Omron Sysmac Studio project PC與TCP Socket測試_5 (Sysmac Studio 1.1.7.20, StandardProject)

# Controller new_Controller_0: NJ501-1300 version 1.10
Units and slaves: 電源 : NJ-Px3001; CPU : NJ501-1300
Axis X, settings changed from default: UnitsConversion=EnumElement2, UnitsNumerator=1048576, UnitsDenominator=5, MaxVelocity=250, MaxJogVelocity=250, HomingMode=BackupAndProximitySignalOff, StartDirection=NegativeDirection, OriginInputDetectionDirection=NegativeDirection, HomingVelocity=50, HomingApproachVelocity=25, CompensationVelocity=25
Axis Y, settings changed from default: AxisNumber=1, UnitsConversion=EnumElement2, UnitsNumerator=1048576, UnitsDenominator=5, MaxVelocity=250, MaxJogVelocity=250, HomingMode=BackupAndProximitySignalOff, StartDirection=NegativeDirection, OriginInputDetectionDirection=NegativeDirection, HomingVelocity=50, HomingApproachVelocity=25, CompensationVelocity=25
Axes group XY_Table, settings changed from default: GroupGroupUse=GroupUsingGroup
Task PrimaryTask (priority 4, period or condition 2000): Program0

TYPE Controller_Socket_Input : STRUCT
    Go_Home_Request : BOOL;
    AutoRun_Request : BOOL;
    MoveStop_Request : BOOL;
    FTP_TablePointRead_Request : BOOL;
    X_Axis_Jog_postive : BOOL;
    X_Axis_Jog_Negtive : BOOL;
    Y_Axis_Jog_postive : BOOL;
    Y_Axis_Jog_Negtive : BOOL;
    X_Axis_PTP_Request : BOOL;
    Y_Axis_PTP_Request : BOOL;
    ErrorReset_Request : BOOL;
    X_Axis_PTP_Position : LREAL;
    X_Axis_PTP_Velocity : LREAL;
    Y_Axis_PTP_Position : LREAL;
    Y_Axis_PTP_Velocity : LREAL;
    AuotoRun_Velocity : LREAL;
END_STRUCT END_TYPE
TYPE Controller_Socket_Output : STRUCT
    Go_Home_Complete : BOOL;
    AutoRun_Busy : BOOL;
    FTP_TablePointRead_Complete : BOOL;
    Error : BOOL;
    X_Axis_Current_Position : LREAL;
    X_Axis_Current_Velocity : LREAL;
    Y_Axis_Current_Position : LREAL;
    Y_Axis_Current_Velocity : LREAL;
END_STRUCT END_TYPE
TYPE XY_TABLE_STRUCT : STRUCT
    X_Axis : LREAL;
    Y_Axis : LREAL;
END_STRUCT END_TYPE

VAR_GLOBAL
    Controller_Socket_Input_Instance : Controller_Socket_Input;
    Controller_Socket_Output_Instance : Controller_Socket_Output;
    TS300_Adress : STRING[100] := '192.168.250.2';
    TS300_TCPPort : UINT;
    TS300_Socket : _sSOCKET;
    TS300_TcpStatus : _eCONNECTION_STATE;
    TS300_Connecting : BOOL;
    TS300_SendString : STRING[256];
    TS300_RcvString : STRING[256];
    TS300_SendByte : ARRAY[0..1999] OF Byte;
    TS300_RcvByte : ARRAY[0..1999] OF Byte;
    TS300_SendByte_Num : UINT;
    TS300_SendByte_Num2 : UINT;
    TS300_TCPSend_Trigger : BOOL;
    TS300_TCPSend_Done : BOOL;
    TS300_TCPRcv_Trigger : BOOL;
    TS300_TCPRcv_Done : BOOL;
    TS300_SktClose_Trigger : BOOL;
    X_AxisAutoRunPoints : ARRAY[0..65534] OF LREAL;
    Y_AxisAutoRunPoints : ARRAY[0..65534] OF LREAL;
END_VAR
VAR_GLOBAL CONSTANT
    X : _sAXIS_REF;  (* at MC://_MC_AX[0] *)
    Y : _sAXIS_REF;  (* at MC://_MC_AX[1] *)
    XY_Table : _sGROUP_REF;  (* at MC://_MC_GRP[0] *)
END_VAR

PROGRAM Program0
VAR
    TS300_TCPConnect : SktTCPConnect;
    TS300_SktClearBuf : SktClearBuf;
    TS300_SktGetStatus : SktGetTCPStatus;
    TS300_SktTCPSend_Instance01 : SktTCPSend;
    TS300_SktTCPRcv_Instance01 : SktTCPRcv;
    TS300_SktClose_Instance01 : SktClose;
    TS300_Connect_Start : BOOL;
    TS300_SktTCPAccept_instance01 : SktTCPAccept;
    SrcTcpPort_TS300 : UINT;
    TCPAccept_Triiger : BOOL;
    Test001 : BOOL;
    TS300_TCPAccept : SktTCPAccept;
    RcvSize : UINT;
    Test002 : BOOL;
    TON_001 : TON;
    TcpStatusNum : DINT;
    TON_002 : TON;
    XY_AutoRunPoints_Read_FB : SDCard_LREAL_Read;
    XY_TablePointsCounts : UINT;
    X_Power_FB : MC_Power;
    Y_Power_FB : MC_Power;
    X_Home_FB : MC_Home;
    Y_Home_FB : MC_Home;
    X_Jog_FB : MC_MoveJog;
    Y_Jog_FB : MC_MoveJog;
    X_Jog_NegativeEnable : BOOL;
    Y_Jog_NegativeEnable : BOOL;
    X_PTPAbs_FB : MC_MoveAbsolute;
    Y_PTPAbs_FB : MC_MoveAbsolute;
    X_STOP_FB : MC_Stop;
    Y_STOP_FB : MC_Stop;
    XY_TableStop_FB : MC_GroupStop;
    X_AxisReset_FB : MC_Reset;
    Y_AxisReset_FB : MC_Reset;
    XY_TableReset_FB : MC_GroupReset;
    XY_TableGroupEnable_FB : MC_GroupEnable;
    XY_TableMoveAbs_FB : ARRAY[0..1] OF MC_MoveLinearAbsolute;
    XY_TablePositionPoints : ARRAY[0..3] OF LREAL;
    Flag : ARRAY[0..1] OF BOOL;
    index : UINT;
    XY_TableGroupDisable_FB : MC_GroupDisable;
    XY_TableGroupDisable_FB_2 : MC_GroupDisable;
END_VAR
VAR_EXTERNAL
    TS300_Adress : STRING[100];
    TS300_TCPPort : UINT;
    TS300_Socket : _sSOCKET;
    TS300_TcpStatus : _eCONNECTION_STATE;
    TS300_Connecting : BOOL;
    TS300_SendString : STRING[256];
    TS300_SendByte : ARRAY[0..1999] OF Byte;
    TS300_SendByte_Num : UINT;
    TS300_SendByte_Num2 : UINT;
    TS300_TCPSend_Trigger : BOOL;
    TS300_TCPSend_Done : BOOL;
    TS300_RcvByte : ARRAY[0..1999] OF Byte;
    TS300_TCPRcv_Trigger : BOOL;
    TS300_TCPRcv_Done : BOOL;
    TS300_SktClose_Trigger : BOOL;
    TS300_RcvString : STRING[256];
    Controller_Socket_Output_Instance : Controller_Socket_Output;
    Controller_Socket_Input_Instance : Controller_Socket_Input;
    X_AxisAutoRunPoints : ARRAY[0..65534] OF LREAL;
    Y_AxisAutoRunPoints : ARRAY[0..65534] OF LREAL;
END_VAR
VAR_EXTERNAL CONSTANT
    X : _sAXIS_REF;
    Y : _sAXIS_REF;
    _ErrSta : WORD;
    XY_Table : _sGROUP_REF;
    _MC_ErrSta : WORD;
    _MC_ComErrSta : WORD;
END_VAR
VAR
    _e1 : R_TRIG;
    _e2 : R_TRIG;
    _e3 : R_TRIG;
    _e4 : R_TRIG;
    _e5 : R_TRIG;
    _e6 : R_TRIG;
    _e7 : R_TRIG;
    _e8 : R_TRIG;
    _e9 : R_TRIG;
    _e10 : R_TRIG;
    _e11 : R_TRIG;
    _e12 : R_TRIG;
    _e13 : R_TRIG;
    _e14 : R_TRIG;
    _e15 : R_TRIG;
    _e16 : R_TRIG;
    _e17 : R_TRIG;
    _e18 : R_TRIG;
    _e19 : R_TRIG;
    _p20 : BOOL;
    _e21 : R_TRIG;
    _p22 : BOOL;
    _e23 : R_TRIG;
    _e24 : R_TRIG;
    _e25 : R_TRIG;
    _t26 : BOOL;
    _br26_0 : BOOL;
    _e27 : R_TRIG;
    _p28 : BOOL;
    _e29 : R_TRIG;
    _e30 : R_TRIG;
    _p31 : BOOL;
    _e32 : R_TRIG;
END_VAR

(* Section TCP_Socket: ladder, written here as Structured Text *)

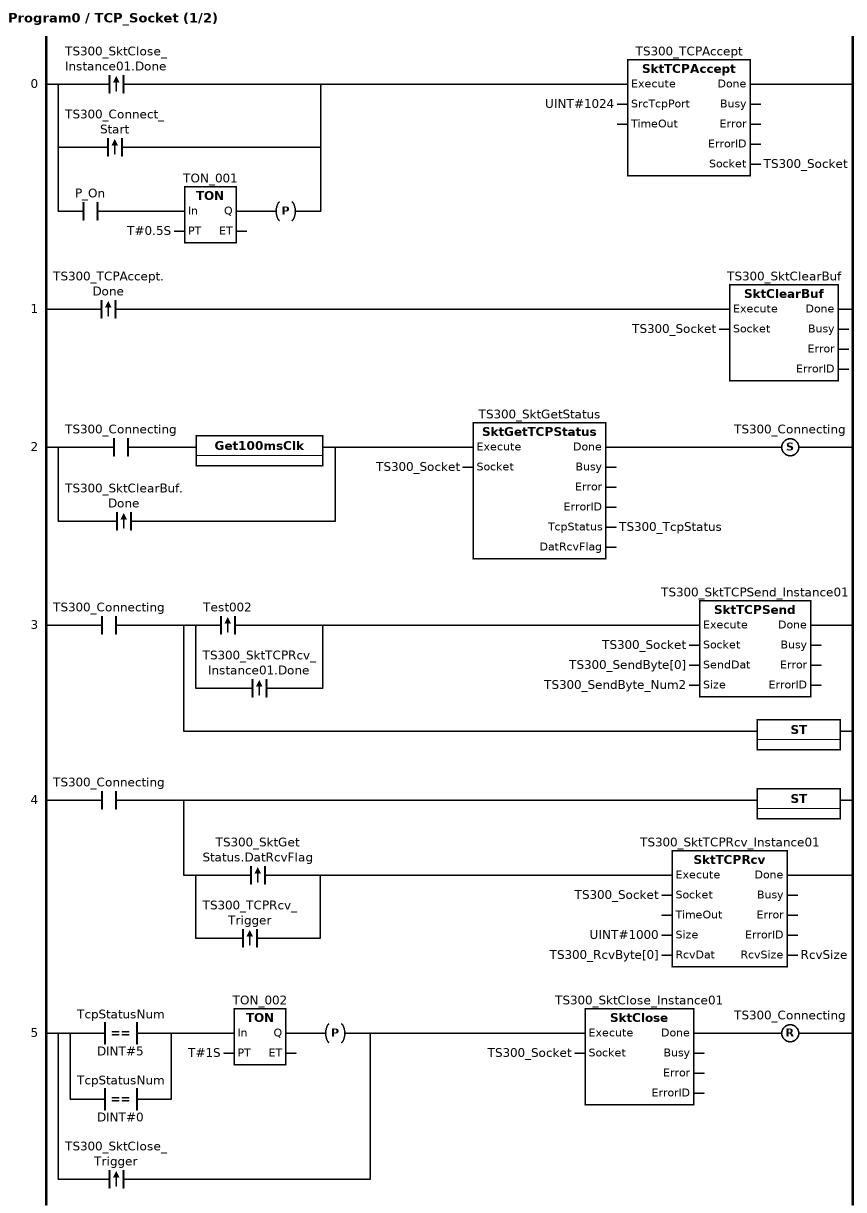
(* Rung 0 *)
_e1(CLK := TS300_SktClose_Instance01.Done);
_e2(CLK := TS300_Connect_Start);
TON_001(In := P_On, PT := T#0.5S);
_e3(CLK := TON_001.Q);
TS300_TCPAccept(Execute := _e1.Q OR _e2.Q OR _e3.Q, SrcTcpPort := UINT#1024, Socket => TS300_Socket);
(* Rung 1 *)
_e4(CLK := TS300_TCPAccept.Done);
TS300_SktClearBuf(Execute := _e4.Q, Socket := TS300_Socket);
(* Rung 2 *)
_e5(CLK := TS300_SktClearBuf.Done);
TS300_SktGetStatus(Execute := (TS300_Connecting AND Get100msClk()) OR _e5.Q, Socket := TS300_Socket, TcpStatus => TS300_TcpStatus);
IF TS300_SktGetStatus.Done THEN TS300_Connecting := TRUE; END_IF;
(* Rung 3 *)
_e6(CLK := Test002);
_e7(CLK := TS300_SktTCPRcv_Instance01.Done);
TS300_SktTCPSend_Instance01(Execute := TS300_Connecting AND (_e6.Q OR _e7.Q), Socket := TS300_Socket, SendDat := TS300_SendByte[0], Size := TS300_SendByte_Num2);
IF TS300_Connecting THEN
    
END_IF;
(* Rung 4 *)
IF TS300_Connecting THEN
    
END_IF;
_e8(CLK := TS300_SktGetStatus.DatRcvFlag);
_e9(CLK := TS300_TCPRcv_Trigger);
TS300_SktTCPRcv_Instance01(Execute := TS300_Connecting AND (_e8.Q OR _e9.Q), Socket := TS300_Socket, Size := UINT#1000, RcvDat := TS300_RcvByte[0], RcvSize => RcvSize);
(* Rung 5 *)
TON_002(In := (TcpStatusNum = DINT#5) OR (TcpStatusNum = DINT#0), PT := T#1S);
_e10(CLK := TON_002.Q);
_e11(CLK := TS300_SktClose_Trigger);
TS300_SktClose_Instance01(Execute := _e10.Q OR _e11.Q, Socket := TS300_Socket);
IF TS300_SktClose_Instance01.Done THEN TS300_Connecting := FALSE; END_IF;

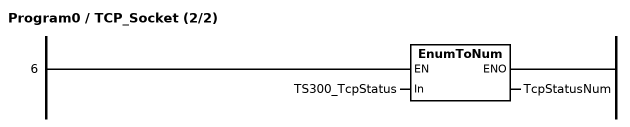
(* Rung 6 *)
TcpStatusNum := EnumToNum(In := TS300_TcpStatus);

(* Section FTP_FileRead: ladder, written here as Structured Text *)

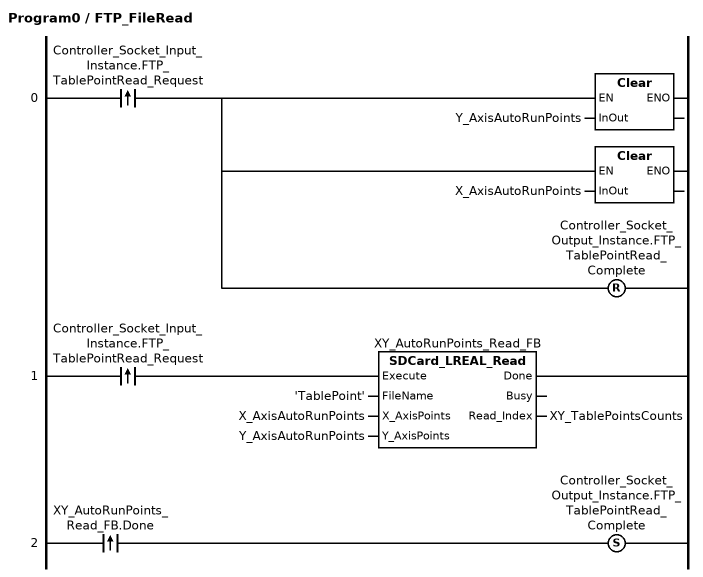
(* Rung 0 *)
_e12(CLK := Controller_Socket_Input_Instance.FTP_TablePointRead_Request);
IF _e12.Q THEN
    Clear(InOut := Y_AxisAutoRunPoints);
    Clear(InOut := X_AxisAutoRunPoints);
    Controller_Socket_Output_Instance.FTP_TablePointRead_Complete := FALSE;
END_IF;
(* Rung 1 *)
_e13(CLK := Controller_Socket_Input_Instance.FTP_TablePointRead_Request);
_e14(CLK := _e13.Q);
XY_AutoRunPoints_Read_FB(Execute := _e14.Q, FileName := 'TablePoint', X_AxisPoints := X_AxisAutoRunPoints, Y_AxisPoints := Y_AxisAutoRunPoints, Read_Index => XY_TablePointsCounts);
(* Rung 2 *)
_e15(CLK := XY_AutoRunPoints_Read_FB.Done);
IF _e15.Q THEN Controller_Socket_Output_Instance.FTP_TablePointRead_Complete := TRUE; END_IF;

(* Section Motion: ladder, written here as Structured Text *)

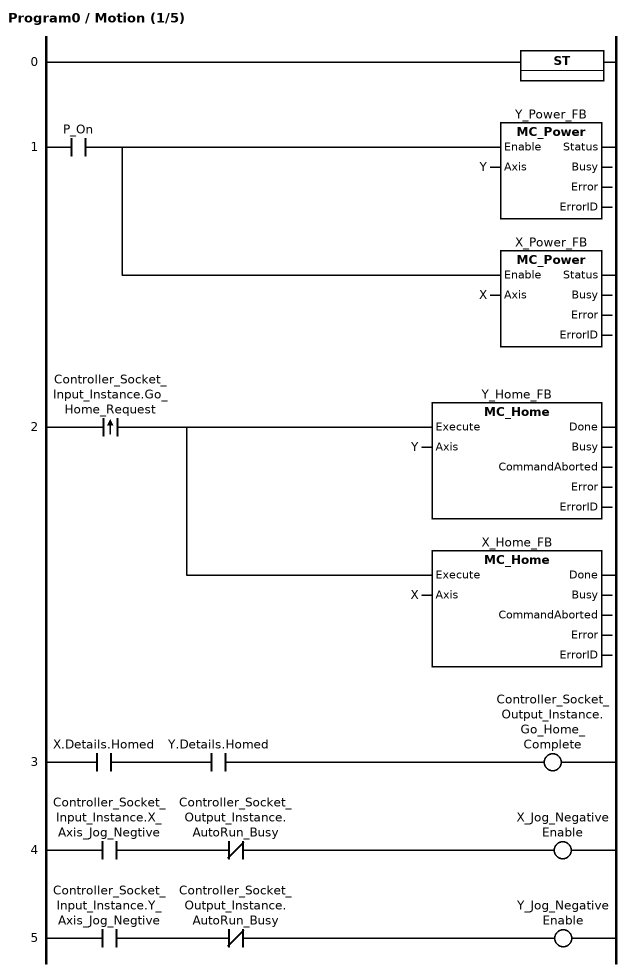
(* Rung 0 *)

(* Rung 1 *)
Y_Power_FB(Enable := P_On, Axis := Y);
X_Power_FB(Enable := P_On, Axis := X);
(* Rung 2 *)
_e16(CLK := Controller_Socket_Input_Instance.Go_Home_Request);
Y_Home_FB(Execute := _e16.Q, Axis := Y);
X_Home_FB(Execute := _e16.Q, Axis := X);
(* Rung 3 *)
Controller_Socket_Output_Instance.Go_Home_Complete := X.Details.Homed AND Y.Details.Homed;
(* Rung 4 *)
X_Jog_NegativeEnable := Controller_Socket_Input_Instance.X_Axis_Jog_Negtive AND NOT Controller_Socket_Output_Instance.AutoRun_Busy;
(* Rung 5 *)
Y_Jog_NegativeEnable := Controller_Socket_Input_Instance.Y_Axis_Jog_Negtive AND NOT Controller_Socket_Output_Instance.AutoRun_Busy;

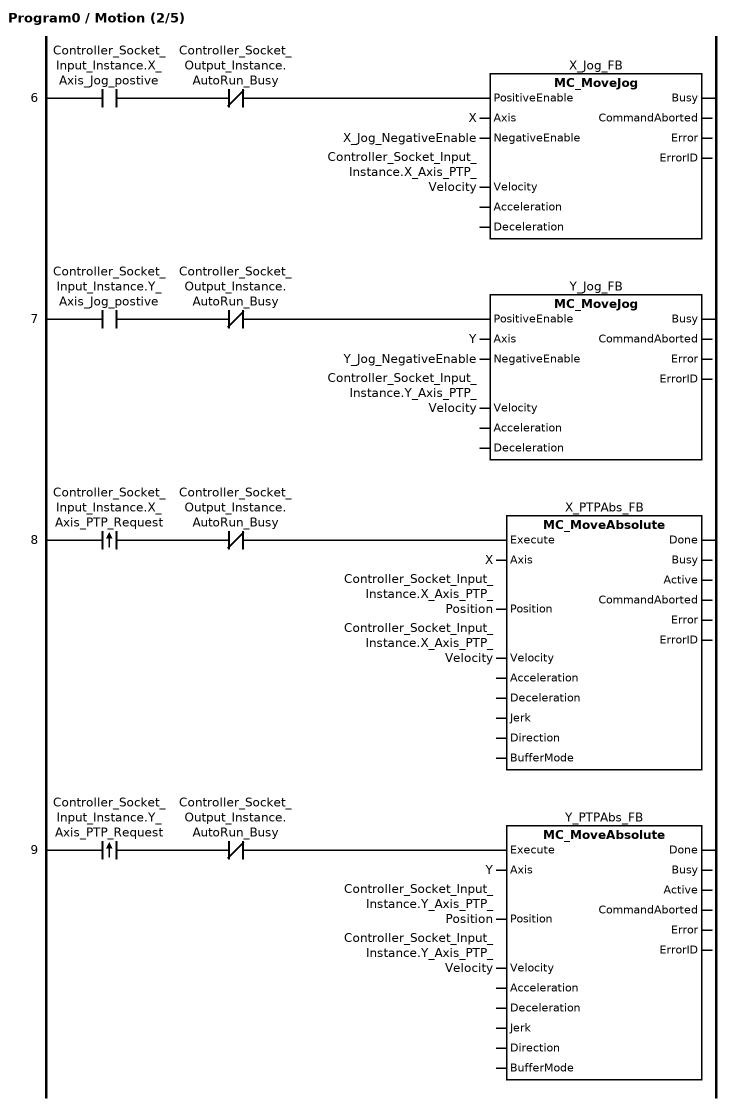
(* Rung 6 *)
X_Jog_FB(PositiveEnable := Controller_Socket_Input_Instance.X_Axis_Jog_postive AND NOT Controller_Socket_Output_Instance.AutoRun_Busy, Axis := X, NegativeEnable := X_Jog_NegativeEnable, Velocity := Controller_Socket_Input_Instance.X_Axis_PTP_Velocity);
(* Rung 7 *)
Y_Jog_FB(PositiveEnable := Controller_Socket_Input_Instance.Y_Axis_Jog_postive AND NOT Controller_Socket_Output_Instance.AutoRun_Busy, Axis := Y, NegativeEnable := Y_Jog_NegativeEnable, Velocity := Controller_Socket_Input_Instance.Y_Axis_PTP_Velocity);
(* Rung 8 *)
_e17(CLK := Controller_Socket_Input_Instance.X_Axis_PTP_Request);
X_PTPAbs_FB(Execute := _e17.Q AND NOT Controller_Socket_Output_Instance.AutoRun_Busy, Axis := X, Position := Controller_Socket_Input_Instance.X_Axis_PTP_Position, Velocity := Controller_Socket_Input_Instance.X_Axis_PTP_Velocity);
(* Rung 9 *)
_e18(CLK := Controller_Socket_Input_Instance.Y_Axis_PTP_Request);
Y_PTPAbs_FB(Execute := _e18.Q AND NOT Controller_Socket_Output_Instance.AutoRun_Busy, Axis := Y, Position := Controller_Socket_Input_Instance.Y_Axis_PTP_Position, Velocity := Controller_Socket_Input_Instance.Y_Axis_PTP_Velocity);

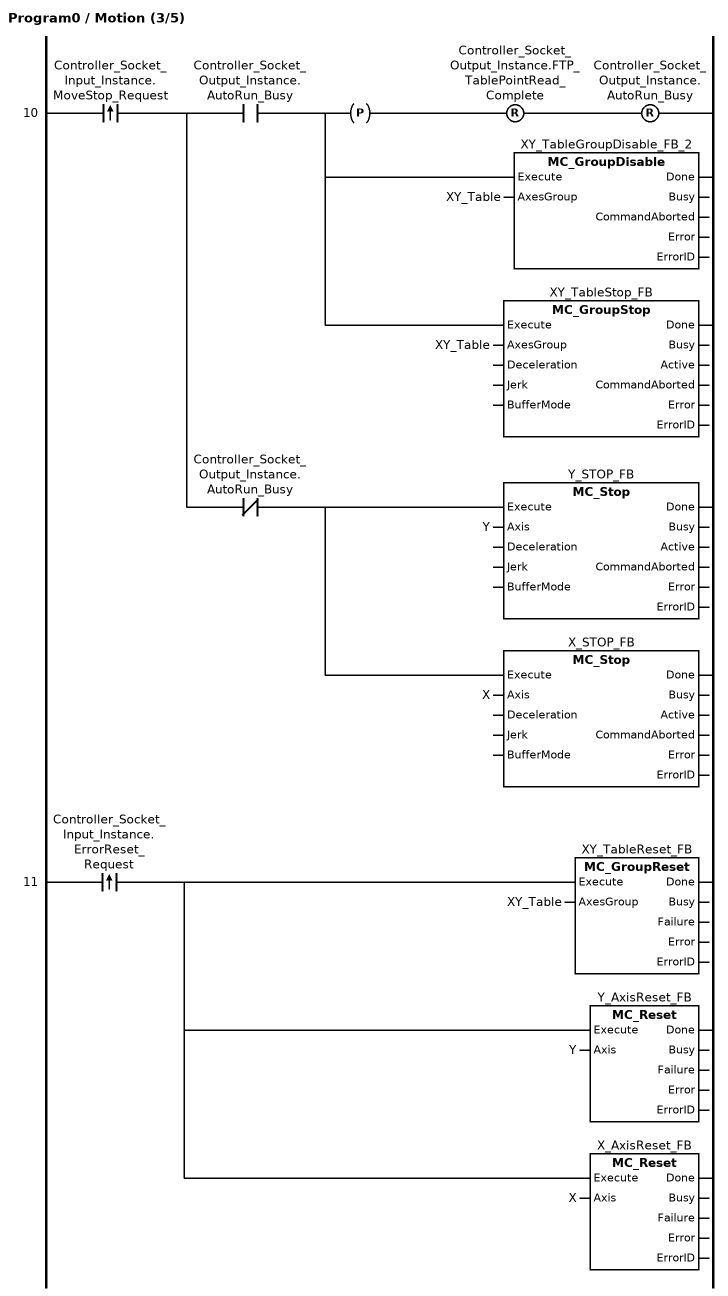
(* Rung 10 *)
_e19(CLK := Controller_Socket_Input_Instance.MoveStop_Request);
_p20 := _e19.Q AND Controller_Socket_Output_Instance.AutoRun_Busy;
_e21(CLK := _p20);
IF _e21.Q THEN
    Controller_Socket_Output_Instance.FTP_TablePointRead_Complete := FALSE;
    Controller_Socket_Output_Instance.AutoRun_Busy := FALSE;
END_IF;
XY_TableGroupDisable_FB_2(Execute := _p20, AxesGroup := XY_Table);
XY_TableStop_FB(Execute := _p20, AxesGroup := XY_Table);
_p22 := _e19.Q AND NOT Controller_Socket_Output_Instance.AutoRun_Busy;
Y_STOP_FB(Execute := _p22, Axis := Y);
X_STOP_FB(Execute := _p22, Axis := X);
(* Rung 11 *)
_e23(CLK := Controller_Socket_Input_Instance.ErrorReset_Request);
XY_TableReset_FB(Execute := _e23.Q, AxesGroup := XY_Table);
Y_AxisReset_FB(Execute := _e23.Q, Axis := Y);
X_AxisReset_FB(Execute := _e23.Q, Axis := X);

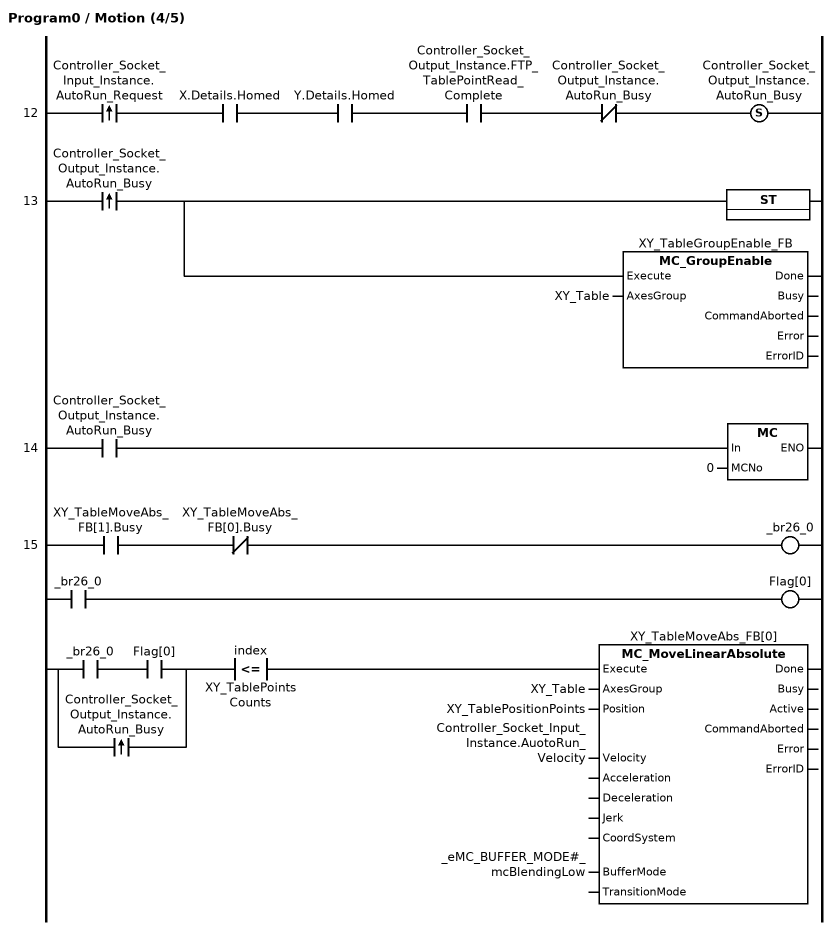
(* Rung 12 *)
_e24(CLK := Controller_Socket_Input_Instance.AutoRun_Request);
IF _e24.Q AND X.Details.Homed AND Y.Details.Homed AND Controller_Socket_Output_Instance.FTP_TablePointRead_Complete AND NOT Controller_Socket_Output_Instance.AutoRun_Busy THEN
    Controller_Socket_Output_Instance.AutoRun_Busy := TRUE;
END_IF;
(* Rung 13 *)
_e25(CLK := Controller_Socket_Output_Instance.AutoRun_Busy);
IF _e25.Q THEN
    
END_IF;
XY_TableGroupEnable_FB(Execute := _e25.Q, AxesGroup := XY_Table);
(* Rung 14 *)
MC(In := Controller_Socket_Output_Instance.AutoRun_Busy, MCNo := 0, ENO => _t26);
(* Rung 15 *)
_br26_0 := XY_TableMoveAbs_FB[1].Busy AND NOT XY_TableMoveAbs_FB[0].Busy;
Flag[0] := _br26_0;
_e27(CLK := Controller_Socket_Output_Instance.AutoRun_Busy);
XY_TableMoveAbs_FB[0](Execute := ((_br26_0 AND Flag[0]) OR _e27.Q) AND (index <= XY_TablePointsCounts), AxesGroup := XY_Table, Position := XY_TablePositionPoints, Velocity := Controller_Socket_Input_Instance.AuotoRun_Velocity, BufferMode := _eMC_BUFFER_MODE#_mcBlendingLow);

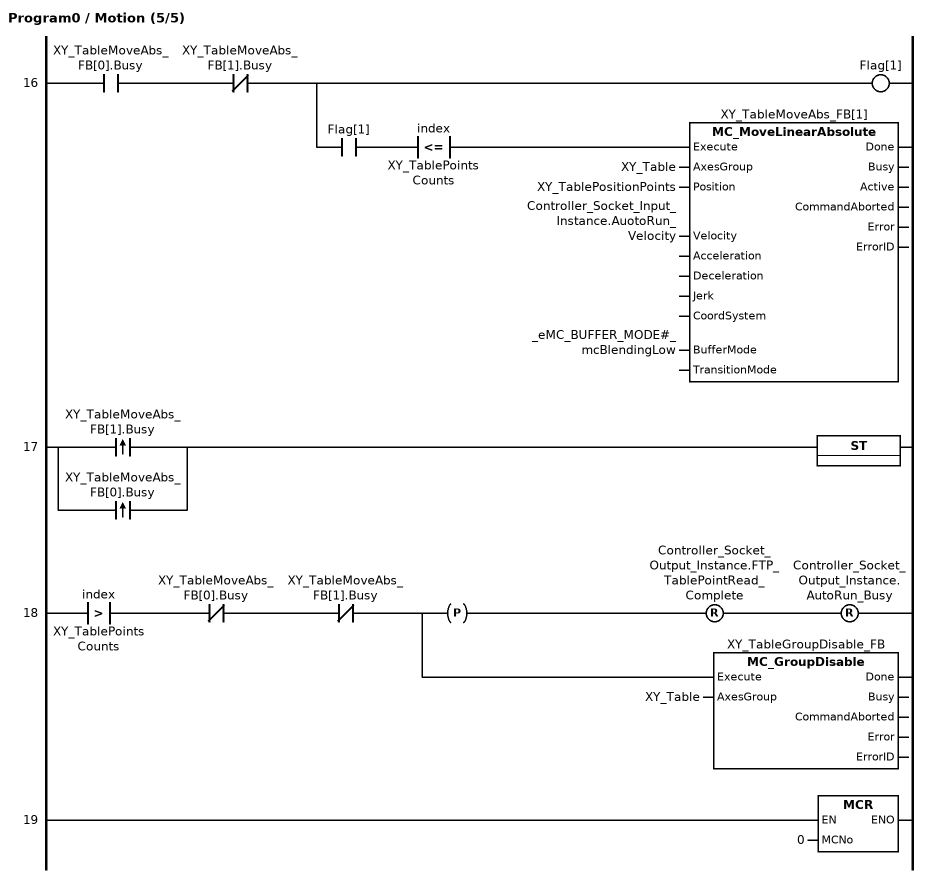
(* Rung 16 *)
_p28 := XY_TableMoveAbs_FB[0].Busy AND NOT XY_TableMoveAbs_FB[1].Busy;
Flag[1] := _p28;
XY_TableMoveAbs_FB[1](Execute := _p28 AND Flag[1] AND (index <= XY_TablePointsCounts), AxesGroup := XY_Table, Position := XY_TablePositionPoints, Velocity := Controller_Socket_Input_Instance.AuotoRun_Velocity, BufferMode := _eMC_BUFFER_MODE#_mcBlendingLow);
(* Rung 17 *)
_e29(CLK := XY_TableMoveAbs_FB[1].Busy);
_e30(CLK := XY_TableMoveAbs_FB[0].Busy);
IF _e29.Q OR _e30.Q THEN
    
END_IF;
(* Rung 18 *)
_p31 := (index > XY_TablePointsCounts) AND NOT XY_TableMoveAbs_FB[0].Busy AND NOT XY_TableMoveAbs_FB[1].Busy;
_e32(CLK := _p31);
IF _e32.Q THEN
    Controller_Socket_Output_Instance.FTP_TablePointRead_Complete := FALSE;
    Controller_Socket_Output_Instance.AutoRun_Busy := FALSE;
END_IF;
XY_TableGroupDisable_FB(Execute := _p31, AxesGroup := XY_Table);
(* Rung 19 *)
MCR(MCNo := 0);
END_PROGRAM

FUNCTION_BLOCK SDCard_LREAL_Read
VAR
    SDCard_Ready : BOOL;
    FileName_All : STRING[105];
    FileRead_Ini : BOOL;
    FileRead_Busy : BOOL;
    FileRead_Stage : UINT;
    FileRead_Index : UINT;
    FileRead_FID : DWORD;
    FileRead_FileOpen : FileOpen;
    FileRead_FileSeek : FileSeek;
    FileRead_Fileget : FileGets;
    FileGet_String : STRING[256];
    XY_TableStruct : XY_TABLE_STRUCT;
    FileRead_FileClose : FileClose;
    R_TRIG_instance : R_TRIG;
END_VAR
VAR_INPUT
    FileName : STRING[100];
    Execute : BOOL (* edge UpDirection *);
END_VAR
VAR_IN_OUT
    X_AxisPoints : ARRAY[0..65534] OF LREAL;
    Y_AxisPoints : ARRAY[0..65534] OF LREAL;
END_VAR
VAR_OUTPUT
    Done : BOOL;
    Busy : BOOL;
    Read_Index : UINT;
END_VAR
VAR_EXTERNAL CONSTANT
    _Card1Ready : BOOL;
END_VAR
SDCard_Ready := _Card1Ready;                                  // _Card1Ready為系統變數實際偵測NJ上是否有抓到插入的SD Card.
FileName_All := CONCAT( FileName , '.CSV');            //功能：結合File_Name(指定讀取檔名)與'.CSV'

//**********************************************************************************************************************************
//*   CSV檔案讀取程式                                                                                                                                                                    *
//**********************************************************************************************************************************
//Execute            為 讀取CSV檔的『觸發BOOL變數』。
//FileRead_Ini     為 讀取CSV檔程式：初始化程序執行中的旗標。
//FileRead_Busy  為 讀取CSV檔程式：讀取資料程序執行中的旗標。 

IF (Execute = TRUE) AND (FileRead_Ini = FALSE) AND (FileRead_Busy = FALSE)  AND (SDCard_Ready)THEN
	FileRead_Ini := TRUE;
	FileRead_Busy := TRUE;
END_IF;

IF (FileRead_Ini = TRUE) THEN
	FileRead_FileOpen( Execute := FALSE);
	FileRead_FileSeek(Execute := FALSE);
	FileRead_Fileget(Execute := FALSE);
	FileRead_FileClose(Execute := FALSE);
	FileRead_Stage := UINT#1;                            //執行步驟流程碼. (步驟1~50) 
	FileRead_Index := UINT#0;                            //Member1 ~ Member2讀取的Size
	FileRead_Ini := FALSE;
END_IF;

IF (FileRead_Busy = TRUE) THEN
	CASE FileRead_Stage OF

		1:
		    FileRead_FileOpen( Execute := TRUE , FileName := FileName_All , Mode :=_READ_EXIST , FileID => FileRead_FID);
			
			IF (FileRead_FileOpen.Done = TRUE) THEN
				FileRead_Stage := 2;
			END_IF;
			IF (FileRead_FileOpen.Error = TRUE) THEN
				FileRead_Stage := 50;
			END_IF;
			
		2:
		    FileRead_FileSeek( Execute := TRUE , FileID := FileRead_FID , Offset := DINT#0 , Origin := _SEEK_SET );
			
			IF (FileRead_FileSeek.Done = TRUE) THEN
				FileRead_Stage := 3;
			END_IF;
			IF (FileRead_FileSeek.Error = TRUE) THEN
				FileRead_Stage := 50;
			END_IF;		
			
		3:
(*********************************寫入使用者定義讀取變數數量  程序*********************************)
(* i1為計數讀取變數數量之Index
    i2為計算加總後的FilePut_String字串數量*)
	 FileRead_FileGet(Execute := TRUE , FileID := FileRead_FID , TrimLF := TRUE );
			
			IF ( FileRead_FileGet.Done = TRUE) THEN
	            FileGet_String := FileRead_FileGet.Out;    //取得SD卡中指定的檔案裡面的一行文字串。
				SubDelimiter(FileGet_String , XY_TableStruct , _COMMA);
				
				X_AxisPoints[FileRead_Index] := XY_TableStruct.X_Axis;
				Y_AxisPoints[FileRead_Index] := XY_TableStruct.Y_Axis;
				
				FileRead_Index := FileRead_Index +1;
				
			    IF (FileRead_FileGet.EOF = FALSE)  THEN
				    FileRead_FileGet(Execute := FALSE );
				ELSE
				    FileRead_Stage := 4;
				END_IF;
			END_IF;
			
			IF (FileRead_FileGet.Error = TRUE ) THEN
				 FileRead_Stage :=50;
			END_IF;
			
		4:
			FileRead_FileClose(Execute := TRUE , FileID := FileRead_FID );
			
			IF (FileRead_FileClose.Done = TRUE ) THEN
				 FileRead_Busy := FALSE;
			END_IF;
			IF (FileRead_FileClose.Error = TRUE ) THEN
				 FileRead_Stage :=50;
			END_IF;
			
		50:
		     FileRead_Busy := FALSE;			 


	END_CASE;
END_IF;

(*Function Block狀態顯示*)
R_TRIG_instance(FileRead_FileClose.Done , Done);
Busy :=  FileRead_Busy;
Read_Index := FileRead_Index -1;
END_FUNCTION_BLOCK